{library PUBLIC}
(* Position number type *)
TYPE PositionType : INT(1..9);
END_TYPE

(* stored: Version 1.1.0.1, ProductVersion 3.1.4024.2
   EnumerationTextList PositionType: Id {f95a2729-eb90-46dd-9f18-e6e36c3a388f} *)
